(* IEC 61131-3 sources: programs/VI-54/VI-54_20171205/VI-54_20171205/Stations/Screen/LseClass170718/Class/RecipeName, 1 file *)

(* ---- RecipeName.st ---- *)
(*!
<Class
	Name               = "RecipeName"
	Revision           = "0.0"
	RealtimeTask       = "false"
	CyclicTask         = "false"
	BackgroundTask     = "false"
	Sigmatek           = "false"
	OSInterface        = "false"
	HighPriority       = "false"
	Automatic          = "false"
	UpdateMode         = "Prescan"
	SharedCommandTable = "true"
	Objectsize         = "(360,300)">
	<Channels>
		<Server Name="R_Date" Visualized="true" Remotely="true" Initialize="true" WriteProtected="false" Retentive="false" Comment="use this channel to access the string functions"/>
		<Server Name="R_Name" Visualized="true" Remotely="true" Initialize="true" WriteProtected="false" Retentive="false" Comment="use this channel to access the string functions"/>
		<Server Name="R_Time" Visualized="true" Remotely="true" Initialize="true" WriteProtected="false" Retentive="false" Comment="use this channel to access the string functions"/>
		<Server Name="RecipeNbr" Visualized="true" Initialize="false" WriteProtected="true" Retentive="false"/>
		<Client Name="Chain" Required="false" Internal="false"/>
		<Client Name="DateString" Required="true" Internal="true"/>
		<Client Name="NameString" Required="true" Internal="true"/>
		<Client Name="TimeString" Required="true" Internal="true"/>
	</Channels>
	<Network Name="RecipeName">
		<!-- List of Components in this network -->
		<Components>
			<Object
				Name       = "DateString"
				Class      = "String"
				Position   = "(240,360)"
				Visualized = "true"
				Remotely   = "true">
				<Channels>
					<Server Name="Data"/>
					<Client Name="SingleRealloc" Value="1"/>
				</Channels>
			</Object>
			<Object
				Name       = "NameString"
				Class      = "String"
				Position   = "(240,210)"
				Visualized = "true"
				Remotely   = "true">
				<Channels>
					<Server Name="Data"/>
					<Client Name="SingleRealloc" Value="1"/>
				</Channels>
			</Object>
			<Object
				Name       = "TimeString"
				Class      = "String"
				Position   = "(240,510)"
				Visualized = "true"
				Remotely   = "true">
				<Channels>
					<Server Name="Data"/>
					<Client Name="SingleRealloc" Value="1"/>
				</Channels>
			</Object>
		</Components>
		<Comments>
		</Comments>
		<!-- List of Connections in this network -->
		<Connections>
			<Connection Source="this.NameString" Destination="NameString.Data"/>
			<Connection Source="this.DateString" Destination="DateString.Data"/>
			<Connection Source="this.TimeString" Destination="TimeString.Data"/>
			<Connection Source="this.R_Name" Destination="NameString.Data" Vertices="(968,270),(796,300),"/>
			<Connection Source="this.R_Date" Destination="DateString.Data" Vertices="(968,330),(796,450),"/>
			<Connection Source="this.R_Time" Destination="TimeString.Data" Vertices="(968,390),(796,600),"/>
		</Connections>
		<!-- Headerfiles -->
		<Options>
		</Options>
	</Network>
</Class>
*)
RecipeName : CLASS
  //Servers:
	RecipeNbr 	: SvrChCmd_DINT;
	R_Name 	: SvrCh_UDINT;
	R_Date 	: SvrCh_UDINT;
	R_Time 	: SvrCh_UDINT;
  //Clients:
	Chain 	: CltChCmd_RecipeName;
	NameString 	: CltChCmd_String;
	DateString 	: CltChCmd_String;
	TimeString 	: CltChCmd_String;
  //Variables:
		TextName 	: DINT;
  //Functions:

	FUNCTION GLOBAL MyInit
		VAR_INPUT
			Number 	: DINT;
		END_VAR
		VAR_OUTPUT
			MaxChain 	: DINT;
		END_VAR;

	FUNCTION GLOBAL WriteNbr
		VAR_INPUT
			Nbr 	: DINT;
		END_VAR;

	FUNCTION GLOBAL WriteName
		VAR_INPUT
			Nbr 	: DINT;
			Name 	: ^CHAR;
			Lenght 	: DINT;
		END_VAR;

	FUNCTION GLOBAL ReadName
		VAR_INPUT
			Nbr 	: DINT;
			Dest 	: ^CHAR;
			MaxSize 	: DINT;
		END_VAR
		VAR_OUTPUT
			Name 	: DINT;
		END_VAR;

	FUNCTION GLOBAL WriteDate
		VAR_INPUT
			Nbr 	: DINT;
			Dates 	: ^CHAR;
			Lenght 	: DINT;
		END_VAR;

	FUNCTION GLOBAL ReadDate
		VAR_INPUT
			Nbr 	: DINT;
			Dest 	: ^CHAR;
			MaxSize 	: DINT;
		END_VAR
		VAR_OUTPUT
			Dates 	: DINT;
		END_VAR;

	FUNCTION GLOBAL WriteTime
		VAR_INPUT
			Nbr 	: DINT;
			Times 	: ^CHAR;
			Lenght 	: DINT;
		END_VAR;

	FUNCTION GLOBAL ReadTime
		VAR_INPUT
			Nbr 	: DINT;
			Dest 	: ^CHAR;
			MaxSize 	: DINT;
		END_VAR
		VAR_OUTPUT
			Times 	: DINT;
		END_VAR;
  //Tables:
	FUNCTION @STD
		VAR_OUTPUT
			ret_code	: CONFSTATES;
		END_VAR;
	FUNCTION GLOBAL TAB @CT_;
END_CLASS;

#pragma using String

FUNCTION GLOBAL RecipeName::MyInit
	VAR_INPUT
		Number 	: DINT;
	END_VAR
	VAR_OUTPUT
		MaxChain 	: DINT;
	END_VAR

  RecipeNbr := Number;

  if IsClientConnected(#Chain) then
    MAxChain := Chain.MyInit(Number:= RecipeNbr + 1);
  else
    MaxChain := RecipeNbr;
  end_if;

END_FUNCTION

FUNCTION GLOBAL RecipeName::WriteNbr
	VAR_INPUT
		Nbr 	: DINT;
	END_VAR

  RecipeNbr := Nbr;

END_FUNCTION

FUNCTION GLOBAL RecipeName::WriteName
	VAR_INPUT
		Nbr 	: DINT;
		Name 	: ^CHAR;
		Lenght 	: DINT;
	END_VAR

  if Nbr = RecipeNbr then
    NameString.WriteDataOff(udLen:= to_Udint(Lenght),
                            udOff:= 0,
                            pData:= Name);
  elsif IsClientConnected(#Chain) then
    Chain.WriteName(Nbr:= Nbr, Name:= Name, Lenght:= Lenght);
  end_if;

END_FUNCTION

FUNCTION GLOBAL RecipeName::ReadName
	VAR_INPUT
		Nbr 	: DINT;
		Dest 	: ^CHAR;
		MaxSize 	: DINT;
	END_VAR
	VAR_OUTPUT
		Name 	: DINT;
	END_VAR

  if Nbr = RecipeNbr then
    Name := to_dint(NameString.ReadDataOff(udOff:= 0, pData:= Dest, udMax:= to_udint(MaxSize)));
  elsif IsClientConnected(#Chain) then
    Name := Chain.ReadName(Nbr:= Nbr, Dest:= Dest, MaxSize:= MaxSize);
  end_if;

END_FUNCTION

FUNCTION GLOBAL RecipeName::WriteDate
	VAR_INPUT
		Nbr 	: DINT;
		Dates 	: ^CHAR;
		Lenght 	: DINT;
	END_VAR

  if Nbr = RecipeNbr then
    DateString.WriteDataOff(udLen:= to_Udint(Lenght),
                            udOff:= 0,
                            pData:= Dates);
  elsif IsClientConnected(#Chain) then
    Chain.WriteDate(Nbr:= Nbr, Dates:= Dates, Lenght:= Lenght);
  end_if;

END_FUNCTION

FUNCTION GLOBAL RecipeName::ReadDate
	VAR_INPUT
		Nbr 	: DINT;
		Dest 	: ^CHAR;
		MaxSize 	: DINT;
	END_VAR
	VAR_OUTPUT
		Dates 	: DINT;
	END_VAR

  if Nbr = RecipeNbr then
    Dates := to_dint(DateString.ReadDataOff(udOff:= 0, pData:= Dest, udMax:= to_udint(MaxSize)));
  elsif IsClientConnected(#Chain) then
    Dates := Chain.ReadDate(Nbr:= Nbr, Dest:= Dest, MaxSize:= MaxSize);
  end_if;

END_FUNCTION

FUNCTION GLOBAL RecipeName::WriteTime
	VAR_INPUT
		Nbr 	: DINT;
		Times 	: ^CHAR;
		Lenght 	: DINT;
	END_VAR

  if Nbr = RecipeNbr then
    TimeString.WriteDataOff(udLen:= to_Udint(Lenght),
                            udOff:= 0,
                            pData:= Times);
  elsif IsClientConnected(#Chain) then
    Chain.WriteTime(Nbr:= Nbr, Times:= Times, Lenght:= Lenght);
  end_if;

END_FUNCTION

FUNCTION GLOBAL RecipeName::ReadTime
	VAR_INPUT
		Nbr 	: DINT;
		Dest 	: ^CHAR;
		MaxSize 	: DINT;
	END_VAR
	VAR_OUTPUT
		Times 	: DINT;
	END_VAR

  if Nbr = RecipeNbr then
    Times := to_dint(TimeString.ReadDataOff(udOff:= 0, pData:= Dest, udMax:= to_udint(MaxSize)));
  elsif IsClientConnected(#Chain) then
    Times := Chain.ReadTime(Nbr:= Nbr, Dest:= Dest, MaxSize:= MaxSize);
  end_if;

END_FUNCTION
